Staubli VAL3: CUTSPACE.pgx

public program CutSpace(string x_sStrIn, string& x_sStrOut)
begin
  //删除数据字符串中最后的空格
  if x_sStrIn!=""
    while right(x_sStrIn,1)==" "
      x_sStrIn=delete(x_sStrIn,1,len(x_sStrIn)-1)
    endWhile
  endIf
  x_sStrOut=x_sStrIn
  //
end
